(* Logix 5000 project; controller ACMI_PLC vendor 1 type 14 code 101 rev 19.11; software revision 19.01; part 9 of 9 *)
(* tags used below, declared in another part *)
   ACMI_ST1_QAB_VAR : REAL;
   ACMI_ST1_QBA_VAR : REAL;
   ACMI_ST2_QAB_VAR : REAL;
   ACMI_ST2_QBA_VAR : REAL;
   C_AVG : REAL;
   C_HIST : DINT[50];
   C_SUM : DINT;
   C_TOP : SINT;
   CAL_Zero : DINT[50];
   CD_N : SINT;
   CLR_CD : BOOL;
   D_AVG : REAL;
   D_HIST : DINT[50];
   D_SUM : DINT;
   D_TOP : SINT;
   EmptyHist : DINT[31];
   Init_INDX : INT[500];
   Init_Stats : BOOL;
   Proc_ST1AB : BOOL;
   Proc_ST1BA : BOOL;
   Proc_ST2AB : BOOL;
   Proc_ST2BA : BOOL;
   Rbit : BOOL;
   REbit : BOOL;
   SSID : STRING;
   SSID_Exists : INT;
   SSID_Locked : INT;
   ST1_HCntr : REAL;
   ST1_QAB_INDX : INT[500];
   ST1_QAB_INDX_TOP : INT;
   ST1_QBA_INDX : INT[500];
   ST1_QBA_INDX_TOP : INT;
   ST2_HCntr : REAL;
   ST2_QAB_INDX : INT[500];
   ST2_QAB_INDX_TOP : INT;
   ST2_QBA_INDX : INT[500];
   ST2_QBA_INDX_TOP : INT;
   A : DINT;
   Abits : INT;
   ACMI_ADC_BITS : INT[2];
   ACMI_BEAM_DATA : REAL[7];
   ACMI_BEAM_Q : REAL;
   ACMI_BR_ACC : REAL;
   ACMI_BR_LIM : REAL;
   ACMI_CERTIFY : SINT;
   ACMI_FAULT_CODE : DINT;
   ACMI_SR_LIM : REAL;
   ACMI_ST1_QAB : REAL;
   ACMI_ST1_QAB_AVG : REAL;
   ACMI_ST1_QAB_HIST : DINT[31];
   ACMI_ST1_QAB_MAX : REAL;
   ACMI_ST1_QAB_MIN : REAL;
   ACMI_ST1_QAB_STD : REAL;
   ACMI_ST1_QBA : REAL;
   ACMI_ST1_QBA_AVG : REAL;
   ACMI_ST1_QBA_HIST : DINT[31];
   ACMI_ST1_QBA_MAX : REAL;
   ACMI_ST1_QBA_MIN : REAL;
   ACMI_ST1_QBA_STD : REAL;
   ACMI_ST2_QAB : REAL;
   ACMI_ST2_QAB_AVG : REAL;
   ACMI_ST2_QAB_HIST : DINT[31];
   ACMI_ST2_QAB_MAX : REAL;
   ACMI_ST2_QAB_MIN : REAL;
   ACMI_ST2_QAB_STD : REAL;
   ACMI_ST2_QBA : REAL;
   ACMI_ST2_QBA_AVG : REAL;
   ACMI_ST2_QBA_HIST : DINT[31];
   ACMI_ST2_QBA_MAX : REAL;
   ACMI_ST2_QBA_MIN : REAL;
   ACMI_ST2_QBA_STD : REAL;
   ACMI_ST_DATA : REAL[24];
   ACMI_TEMPS : INT[6];
   ACMI_TIMING : SINT;
   ACMI_TO_ACC : REAL;
   B : DINT;
   Bbits : INT;
   Beam_MaxQ : DINT;
   Beam_MinQ : DINT;
   Beam_Q : DINT;
   BR_Stack_MAX : DINT;
   BR_Stack_Sum : DINT;
   FAULT_CODE : DINT;
   HMI_BEAM_Q : REAL;
   HMI_Suppress : BOOL;
   Relay_Error : BOOL;
   RESET_FAULT : ALIAS FOR PointIONet:5:I.Pt01Data;
   ST1_MaxQ : DINT;
   ST1_MinQ : DINT;
   ST1_QAB : DINT;
   ST1_QBA : DINT;
   ST1AB_Size : INT;
   ST1BA_Size : INT;
   ST2_MaxQ : DINT;
   ST2_MinQ : DINT;
   ST2_QAB : DINT;
   ST2_QBA : DINT;
   ST2AB_Size : INT;
   ST2BA_Size : INT;
   TO_Stack_MAX : DINT;
   TO_Stack_Sum : DINT;
   Update_ST1_QAB : BOOL;
   Update_ST1_QBA : BOOL;
   Update_ST2_QAB : BOOL;
   Update_ST2_QBA : BOOL;
(* MainProgram, continued *)

ROUTINE CD_Stats   (* ladder *)
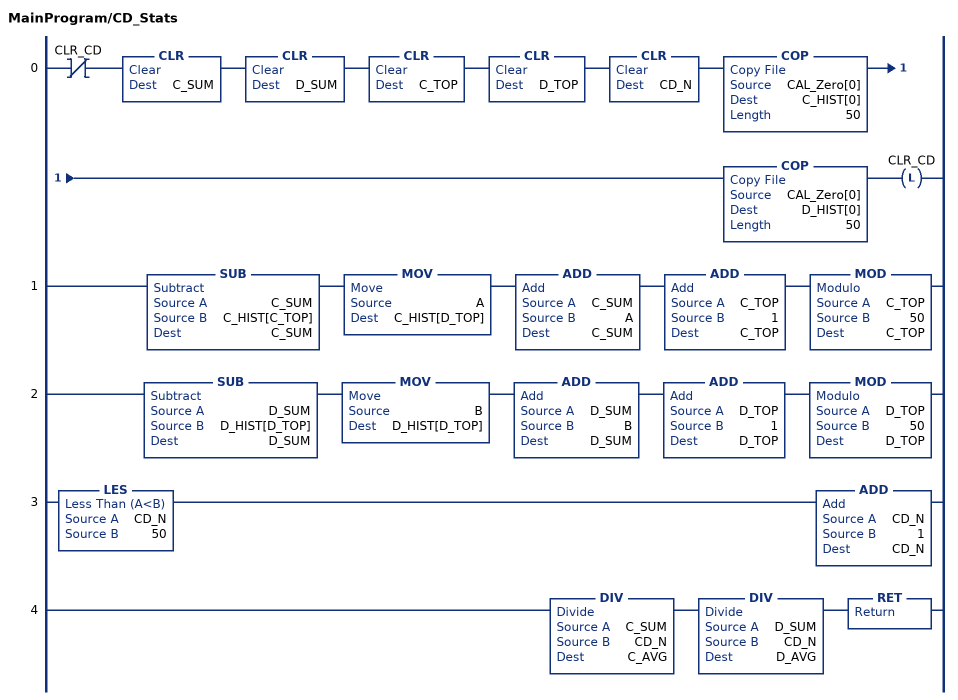
   0: XIO(CLR_CD)CLR(C_SUM)CLR(D_SUM)CLR(C_TOP)CLR(D_TOP)CLR(CD_N)COP(CAL_Zero[0],C_HIST[0],50)COP(CAL_Zero[0],D_HIST[0],50)OTL(CLR_CD);
   1: SUB(C_SUM,C_HIST[C_TOP],C_SUM)MOV(A,C_HIST[D_TOP])ADD(C_SUM,A,C_SUM)ADD(C_TOP,1,C_TOP)MOD(C_TOP,50,C_TOP);
   2: SUB(D_SUM,D_HIST[D_TOP],D_SUM)MOV(B,D_HIST[D_TOP])ADD(D_SUM,B,D_SUM)ADD(D_TOP,1,D_TOP)MOD(D_TOP,50,D_TOP);
   3: LES(CD_N,50)ADD(CD_N,1,CD_N);
   4: DIV(C_SUM,CD_N,C_AVG)DIV(D_SUM,CD_N,D_AVG)RET();
END_ROUTINE

ROUTINE Self_Test_Stats   (* ladder *)
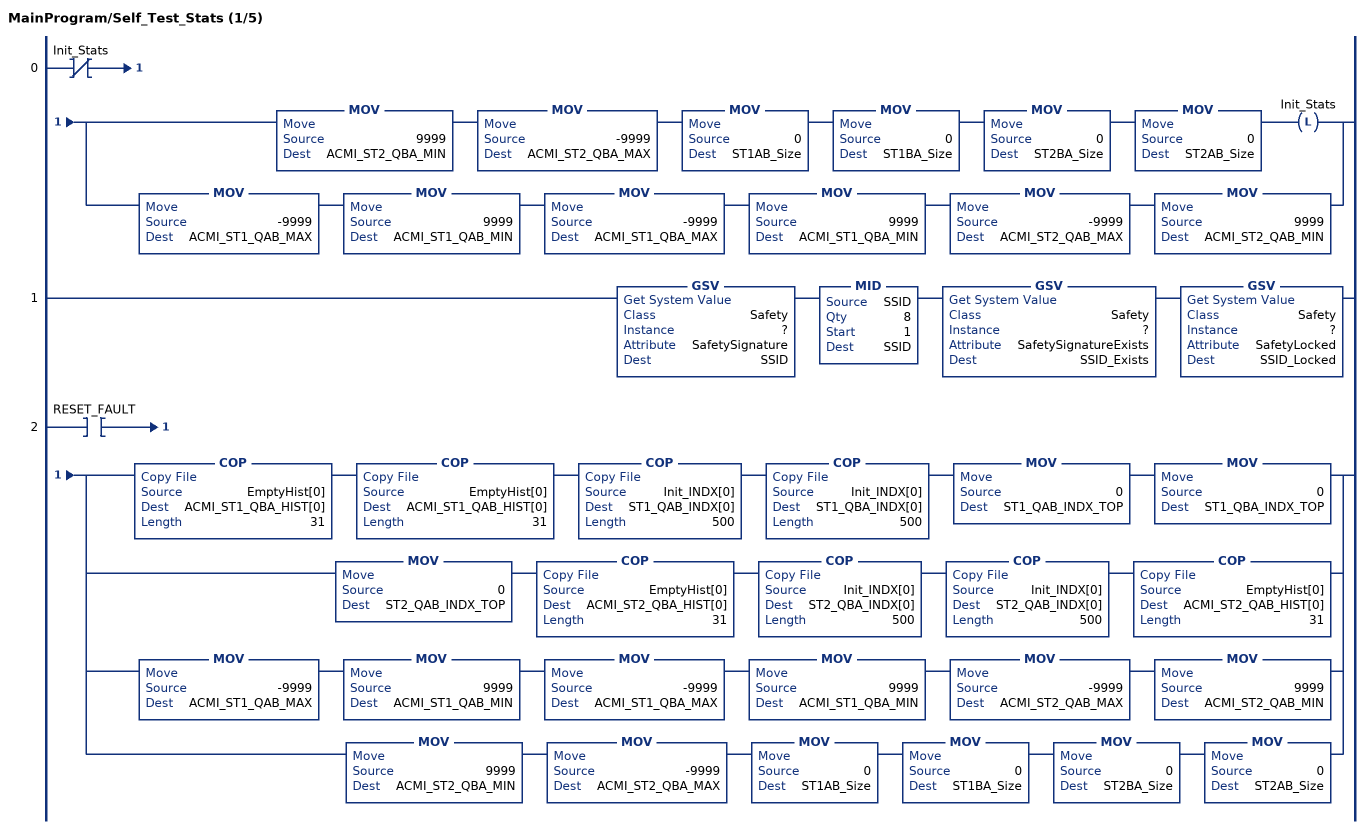
   0: XIO(Init_Stats)[MOV(9999,ACMI_ST2_QBA_MIN) MOV(-9999,ACMI_ST2_QBA_MAX) MOV(0,ST1AB_Size) MOV(0,ST1BA_Size) MOV(0,ST2BA_Size) MOV(0,ST2AB_Size) OTL(Init_Stats) ,MOV(-9999,ACMI_ST1_QAB_MAX) MOV(9999,ACMI_ST1_QAB_MIN) MOV(-9999,ACMI_ST1_QBA_MAX) MOV(9999,ACMI_ST1_QBA_MIN) MOV(-9999,ACMI_ST2_QAB_MAX) MOV(9999,ACMI_ST2_QAB_MIN) ];
   1: GSV(Safety,?,SafetySignature,SSID)MID(SSID,8,1,SSID)GSV(Safety,?,SafetySignatureExists,SSID_Exists)GSV(Safety,?,SafetyLocked,SSID_Locked);
   2: XIC(RESET_FAULT)[COP(EmptyHist[0],ACMI_ST1_QBA_HIST[0],31) COP(EmptyHist[0],ACMI_ST1_QAB_HIST[0],31) COP(Init_INDX[0],ST1_QAB_INDX[0],500) COP(Init_INDX[0],ST1_QBA_INDX[0],500) MOV(0,ST1_QAB_INDX_TOP) MOV(0,ST1_QBA_INDX_TOP) ,MOV(0,ST2_QAB_INDX_TOP) COP(EmptyHist[0],ACMI_ST2_QBA_HIST[0],31) COP(Init_INDX[0],ST2_QBA_INDX[0],500) COP(Init_INDX[0],ST2_QAB_INDX[0],500) COP(EmptyHist[0],ACMI_ST2_QAB_HIST[0],31) ,MOV(-9999,ACMI_ST1_QAB_MAX) MOV(9999,ACMI_ST1_QAB_MIN) MOV(-9999,ACMI_ST1_QBA_MAX) MOV(9999,ACMI_ST1_QBA_MIN) MOV(-9999,ACMI_ST2_QAB_MAX) MOV(9999,ACMI_ST2_QAB_MIN) ,MOV(9999,ACMI_ST2_QBA_MIN) MOV(-9999,ACMI_ST2_QBA_MAX) MOV(0,ST1AB_Size) MOV(0,ST1BA_Size) MOV(0,ST2BA_Size) MOV(0,ST2AB_Size) ];
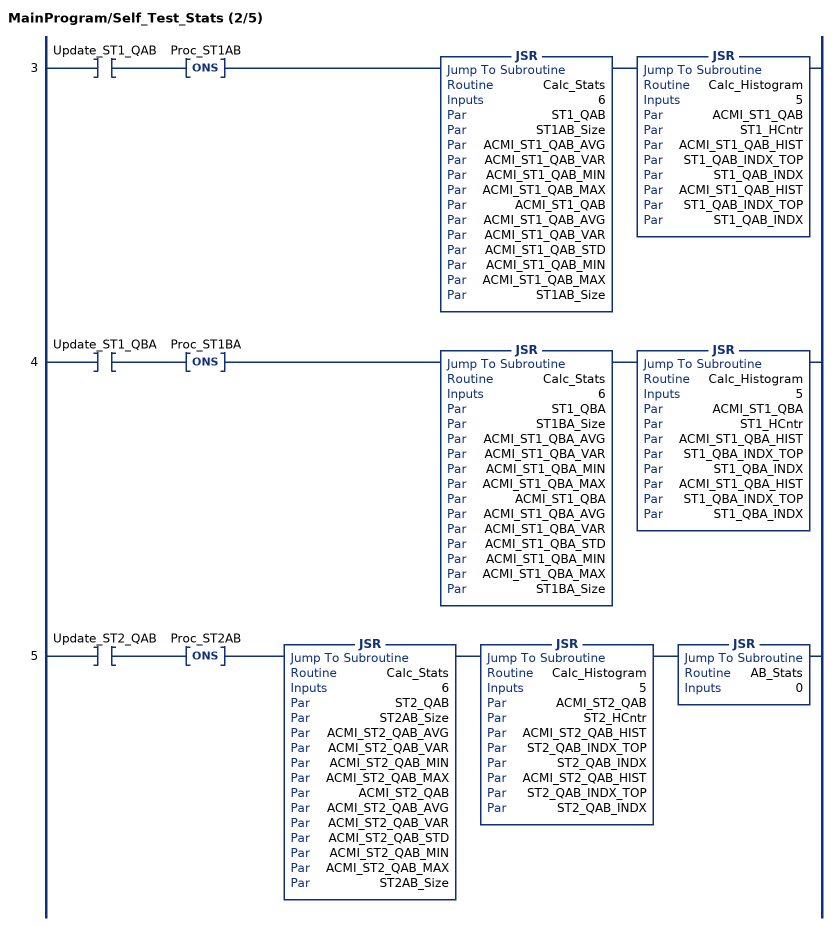
   3: XIC(Update_ST1_QAB)ONS(Proc_ST1AB)JSR(Calc_Stats,6,ST1_QAB,ST1AB_Size,ACMI_ST1_QAB_AVG,ACMI_ST1_QAB_VAR,ACMI_ST1_QAB_MIN,ACMI_ST1_QAB_MAX,ACMI_ST1_QAB,ACMI_ST1_QAB_AVG,ACMI_ST1_QAB_VAR,ACMI_ST1_QAB_STD,ACMI_ST1_QAB_MIN,ACMI_ST1_QAB_MAX,ST1AB_Size)JSR(Calc_Histogram,5,ACMI_ST1_QAB,ST1_HCntr,ACMI_ST1_QAB_HIST,ST1_QAB_INDX_TOP,ST1_QAB_INDX,ACMI_ST1_QAB_HIST,ST1_QAB_INDX_TOP,ST1_QAB_INDX);
   4: XIC(Update_ST1_QBA)ONS(Proc_ST1BA)JSR(Calc_Stats,6,ST1_QBA,ST1BA_Size,ACMI_ST1_QBA_AVG,ACMI_ST1_QBA_VAR,ACMI_ST1_QBA_MIN,ACMI_ST1_QBA_MAX,ACMI_ST1_QBA,ACMI_ST1_QBA_AVG,ACMI_ST1_QBA_VAR,ACMI_ST1_QBA_STD,ACMI_ST1_QBA_MIN,ACMI_ST1_QBA_MAX,ST1BA_Size)JSR(Calc_Histogram,5,ACMI_ST1_QBA,ST1_HCntr,ACMI_ST1_QBA_HIST,ST1_QBA_INDX_TOP,ST1_QBA_INDX,ACMI_ST1_QBA_HIST,ST1_QBA_INDX_TOP,ST1_QBA_INDX);
   5: XIC(Update_ST2_QAB)ONS(Proc_ST2AB)JSR(Calc_Stats,6,ST2_QAB,ST2AB_Size,ACMI_ST2_QAB_AVG,ACMI_ST2_QAB_VAR,ACMI_ST2_QAB_MIN,ACMI_ST2_QAB_MAX,ACMI_ST2_QAB,ACMI_ST2_QAB_AVG,ACMI_ST2_QAB_VAR,ACMI_ST2_QAB_STD,ACMI_ST2_QAB_MIN,ACMI_ST2_QAB_MAX,ST2AB_Size)JSR(Calc_Histogram,5,ACMI_ST2_QAB,ST2_HCntr,ACMI_ST2_QAB_HIST,ST2_QAB_INDX_TOP,ST2_QAB_INDX,ACMI_ST2_QAB_HIST,ST2_QAB_INDX_TOP,ST2_QAB_INDX)JSR(AB_Stats,0);
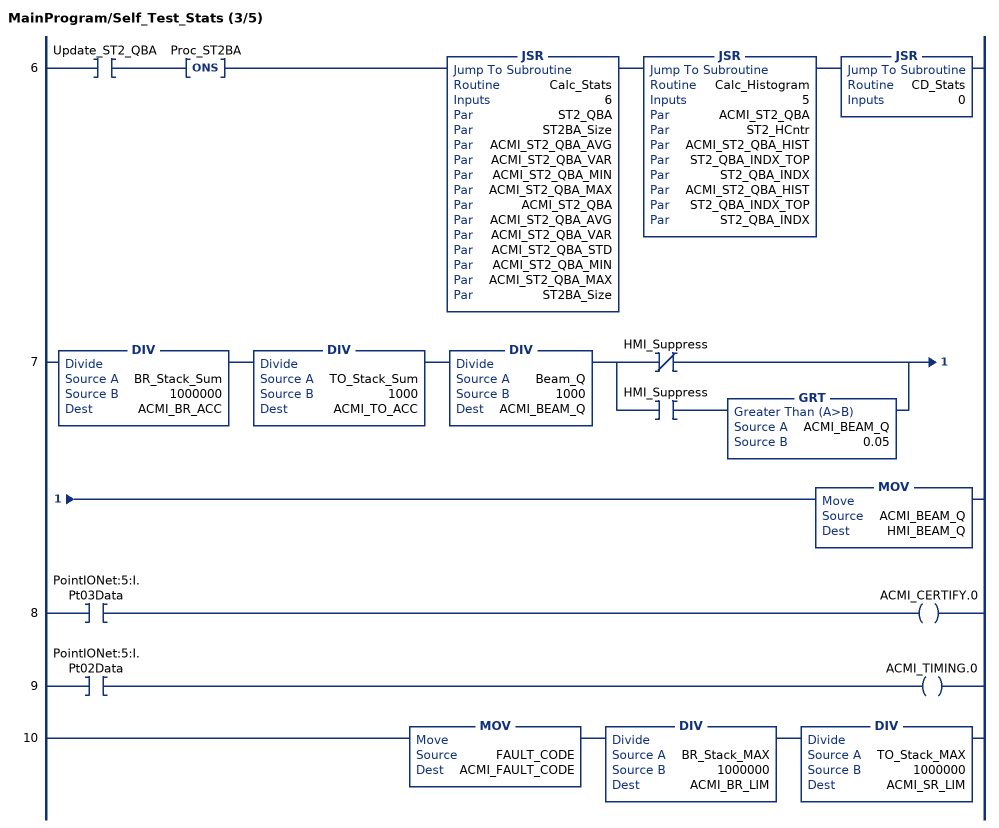
   6: XIC(Update_ST2_QBA)ONS(Proc_ST2BA)JSR(Calc_Stats,6,ST2_QBA,ST2BA_Size,ACMI_ST2_QBA_AVG,ACMI_ST2_QBA_VAR,ACMI_ST2_QBA_MIN,ACMI_ST2_QBA_MAX,ACMI_ST2_QBA,ACMI_ST2_QBA_AVG,ACMI_ST2_QBA_VAR,ACMI_ST2_QBA_STD,ACMI_ST2_QBA_MIN,ACMI_ST2_QBA_MAX,ST2BA_Size)JSR(Calc_Histogram,5,ACMI_ST2_QBA,ST2_HCntr,ACMI_ST2_QBA_HIST,ST2_QBA_INDX_TOP,ST2_QBA_INDX,ACMI_ST2_QBA_HIST,ST2_QBA_INDX_TOP,ST2_QBA_INDX)JSR(CD_Stats,0);
   7: DIV(BR_Stack_Sum,1000000,ACMI_BR_ACC)DIV(TO_Stack_Sum,1000,ACMI_TO_ACC)DIV(Beam_Q,1000,ACMI_BEAM_Q)[XIO(HMI_Suppress) ,XIC(HMI_Suppress) GRT(ACMI_BEAM_Q,0.05) ]MOV(ACMI_BEAM_Q,HMI_BEAM_Q);
   8: XIC(PointIONet:5:I.Pt03Data)OTE(ACMI_CERTIFY.0);
   9: XIC(PointIONet:5:I.Pt02Data)OTE(ACMI_TIMING.0);
   10: MOV(FAULT_CODE,ACMI_FAULT_CODE)DIV(BR_Stack_MAX,1000000,ACMI_BR_LIM)DIV(TO_Stack_MAX,1000000,ACMI_SR_LIM);
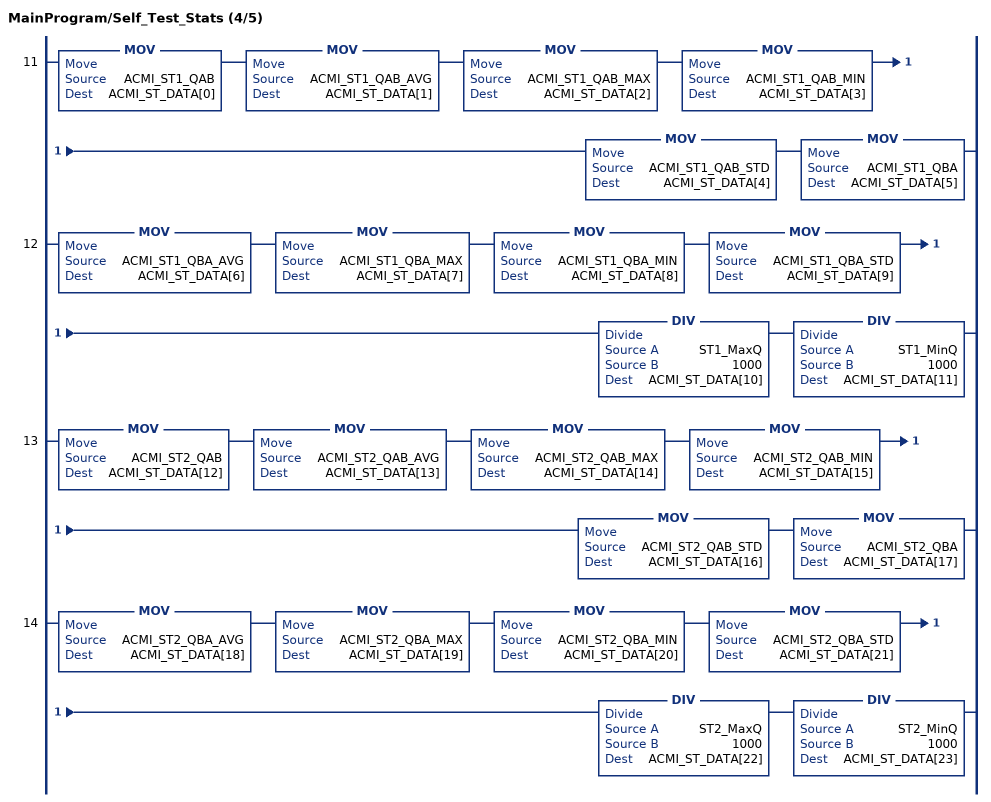
   11: MOV(ACMI_ST1_QAB,ACMI_ST_DATA[0])MOV(ACMI_ST1_QAB_AVG,ACMI_ST_DATA[1])MOV(ACMI_ST1_QAB_MAX,ACMI_ST_DATA[2])MOV(ACMI_ST1_QAB_MIN,ACMI_ST_DATA[3])MOV(ACMI_ST1_QAB_STD,ACMI_ST_DATA[4])MOV(ACMI_ST1_QBA,ACMI_ST_DATA[5]);
   12: MOV(ACMI_ST1_QBA_AVG,ACMI_ST_DATA[6])MOV(ACMI_ST1_QBA_MAX,ACMI_ST_DATA[7])MOV(ACMI_ST1_QBA_MIN,ACMI_ST_DATA[8])MOV(ACMI_ST1_QBA_STD,ACMI_ST_DATA[9])DIV(ST1_MaxQ,1000,ACMI_ST_DATA[10])DIV(ST1_MinQ,1000,ACMI_ST_DATA[11]);
   13: MOV(ACMI_ST2_QAB,ACMI_ST_DATA[12])MOV(ACMI_ST2_QAB_AVG,ACMI_ST_DATA[13])MOV(ACMI_ST2_QAB_MAX,ACMI_ST_DATA[14])MOV(ACMI_ST2_QAB_MIN,ACMI_ST_DATA[15])MOV(ACMI_ST2_QAB_STD,ACMI_ST_DATA[16])MOV(ACMI_ST2_QBA,ACMI_ST_DATA[17]);
   14: MOV(ACMI_ST2_QBA_AVG,ACMI_ST_DATA[18])MOV(ACMI_ST2_QBA_MAX,ACMI_ST_DATA[19])MOV(ACMI_ST2_QBA_MIN,ACMI_ST_DATA[20])MOV(ACMI_ST2_QBA_STD,ACMI_ST_DATA[21])DIV(ST2_MaxQ,1000,ACMI_ST_DATA[22])DIV(ST2_MinQ,1000,ACMI_ST_DATA[23]);
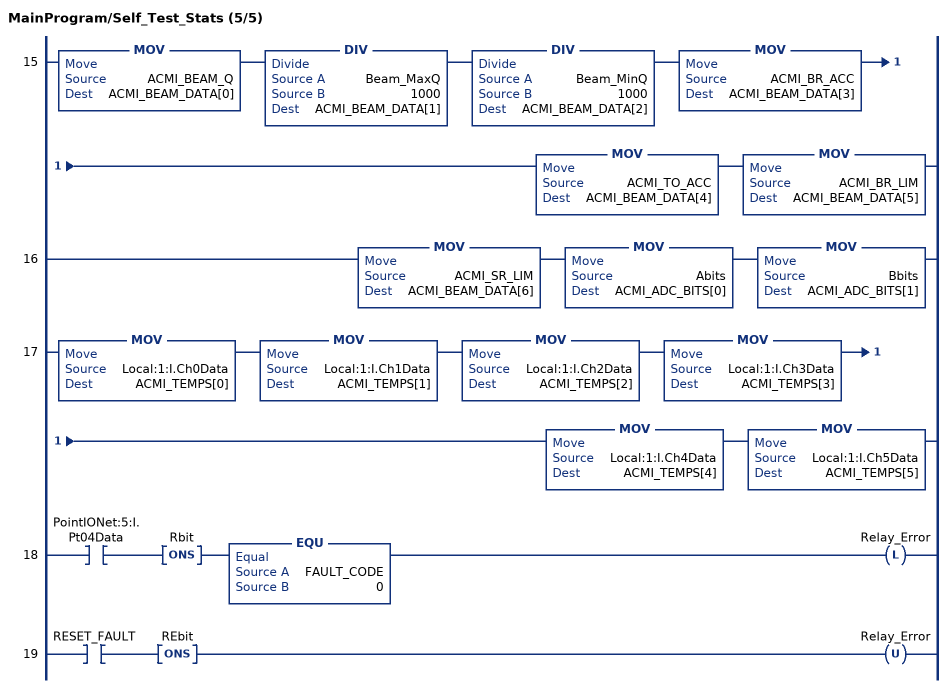
   15: MOV(ACMI_BEAM_Q,ACMI_BEAM_DATA[0])DIV(Beam_MaxQ,1000,ACMI_BEAM_DATA[1])DIV(Beam_MinQ,1000,ACMI_BEAM_DATA[2])MOV(ACMI_BR_ACC,ACMI_BEAM_DATA[3])MOV(ACMI_TO_ACC,ACMI_BEAM_DATA[4])MOV(ACMI_BR_LIM,ACMI_BEAM_DATA[5]);
   16: MOV(ACMI_SR_LIM,ACMI_BEAM_DATA[6])MOV(Abits,ACMI_ADC_BITS[0])MOV(Bbits,ACMI_ADC_BITS[1]);
   17: MOV(Local:1:I.Ch0Data,ACMI_TEMPS[0])MOV(Local:1:I.Ch1Data,ACMI_TEMPS[1])MOV(Local:1:I.Ch2Data,ACMI_TEMPS[2])MOV(Local:1:I.Ch3Data,ACMI_TEMPS[3])MOV(Local:1:I.Ch4Data,ACMI_TEMPS[4])MOV(Local:1:I.Ch5Data,ACMI_TEMPS[5]);
   18: XIC(PointIONet:5:I.Pt04Data)ONS(Rbit)EQU(FAULT_CODE,0)OTL(Relay_Error);
   19: XIC(RESET_FAULT)ONS(REbit)OTU(Relay_Error);
END_ROUTINE
END_PROGRAM
